{attribute 'linkalways'} 
{attribute 'no_explicit_call' := 'This FB is a CLASS and must be accessed using methods or properties'}
{attribute 'enable_dynamic_creation'}
FUNCTION_BLOCK Node_F_VN_AddToContainerElements_UDINT EXTENDS VisionNode
VAR
    nValue : _UDINT(0);
    ipContainer : _ITcVnContainer;
    hrPrev : _HRESULT(S_OK);
    hresult : _HRESULT(S_OK);
END_VAR

METHOD PUBLIC  Clone : I_Node
VAR
    pNode : POINTER TO Node_F_VN_AddToContainerElements_UDINT;
END_VAR
pNode := __NEW(Node_F_VN_AddToContainerElements_UDINT);
Clone := pNode^;
END_METHOD

METHOD FB_init : BOOL
VAR_INPUT
    bInitRetains : BOOL; // if TRUE, the retain variables are initialized (warm start / cold start)
    bInCopyCode : BOOL;  // if TRUE, the instance afterwards gets moved into the copy code (online change)
END_VAR
AddParameter('nValue', nValue);
AddInput('ipContainer', ipContainer);
AddInput('hrPrev', hrPrev);
AddOutput('ipContainer', ipContainer);
AddOutput('hresult',hresult);
END_METHOD

METHOD PROTECTED OnExecute
hresult.Value := F_VN_AddToContainerElements_UDINT(
    nValue := nValue.Value,
    ipContainer := ipContainer.Value,
    hrPrev:= hrPrev.Value);
END_METHOD

METHOD PUBLIC PreExecutionCheck
VAR_INPUT
    Check : I_PreExecutionChecks;
END_VAR
Check.IsTrue(ipContainer.IsValid, 'ipContainer must be a valid container');
Check.IsTrue(ipContainer.IsType(TC_GLOBAL_CONST_LIST.ContainerType_Vector_UDINT), 'ipContainer contains incorrect type');
END_METHOD

END_FUNCTION_BLOCK

(* stored: Version 1.1.0.1, ProductVersion 3.1.4026.13
   POU Node_F_VN_AddToContainerElements_UDINT: Id {3c689135-ea5f-4251-ae89-e8ab0d57fb4e}, SpecialFunc None
   Folder Constructor: Id {78e8314a-36dc-4ece-b66d-2e036b1a5e2b}
   Method Clone: Id {a3170854-5572-4d3e-a7f4-1bb2e5b344b7}
   Method FB_init: Id {4f558769-69b2-45cb-b5c5-4e910d1de128}
   Method OnExecute: Id {7cdd6fba-13fc-4a7c-9158-db3cdaa1f96f}
   Method PreExecutionCheck: Id {5585f74b-b3dc-4843-98c0-8eb62f92e328} *)
